{attribute 'linkalways'} 
{attribute 'no_explicit_call' := 'This FB is a CLASS and must be accessed using methods or properties'}
{attribute 'enable_dynamic_creation'}
FUNCTION_BLOCK FINAL MOD_LINT EXTENDS Node
VAR
	in1 : _LINT(0);
	in2 : _LINT(0);
	out : _LINT(0);
END_VAR

METHOD PUBLIC Clone : I_Node
VAR
	pNode : POINTER TO MOD_LINT;
END_VAR
pNode := __NEW(MOD_LINT);
Clone := pNode^;
END_METHOD

METHOD FB_init : BOOL
VAR_INPUT
	bInitRetains : BOOL; // if TRUE, the retain variables are initialized (warm start / cold start)
	bInCopyCode : BOOL;  // if TRUE, the instance afterwards gets moved into the copy code (online change)
END_VAR
AddInput('in1',THIS^.in1);
AddInput('in2',THIS^.in2);
AddOutput('out', THIS^.out);
END_METHOD

METHOD PROTECTED OnExecute
VAR
END_VAR
out.Value := in1.Value MOD in2.Value;
END_METHOD

END_FUNCTION_BLOCK

(* stored: Version 1.1.0.1, ProductVersion 3.1.4024.15
   POU MOD_LINT: Id {126e67b0-1d21-40b8-9625-a02ad975e5e5}, SpecialFunc None
   Folder Constructor: Id {71e8c60f-af61-42e1-bd1f-22cfd7968a0d}
   Method Clone: Id {b115a8b1-b30b-4499-90ad-67e9ea98d4c9}
   Method FB_init: Id {2e732048-bb0f-4ddb-a8aa-1e5d3d6aff7d}
   Method OnExecute: Id {95e519a0-a4ac-45be-8e37-34476d153291} *)
